DATA_BLOCK "DB"
{ S7_Optimized_Access := 'true' }
    VAR
        aut_y: LREAL;
        i: DINT;
        bol: BOOL;
        col: BYTE;
        firstRun: BOOL;
    END_VAR
BEGIN
    firstRun := TRUE;
END_DATA_BLOCK
